{attribute 'qualified_only'}
{attribute 'strict'}
{attribute 'to_string'}
TYPE AlarmList :
(
	emergency_stop := 1,
	encoder_error,
	approach,
	proximity,
	collision
);
END_TYPE

(* stored: Version 1.1.0.1
   DUT AlarmList: Id {e838e5c6-f57b-4165-8f8f-acd96c37ea14} *)
